FUNCTION TryConvert_TIME_TO_DT : BOOL
VAR_INPUT
	in : TIME;
	out : REFERENCE TO DT;
END_VAR

out := TIME_TO_DT(in);
TryConvert_TIME_TO_DT := TRUE;

END_FUNCTION

(* stored: Version 1.1.0.1, ProductVersion 3.1.4024.12
   POU TryConvert_TIME_TO_DT: Id {936f771a-bff2-4f48-8c20-ab987a484c7c}, SpecialFunc None *)
